(* IEC 61131-3 sources: LabBench/FB, 3 files *)

(* ---- FB_FloatLevelSensorGroup.st ---- *)
(*==============================================================================
    Название:    FB_FloatLevelSensorGroup
    Автор:       Инженер ПЛК
    Дата:        2025-04-26
    Версия:      1.0

    Описание:    Функциональный блок для группы поплавковых датчиков уровня.
                 Группа состоит из трех датчиков, расположенных на различных
                 уровнях в емкости высотой 500 мм:
                 - Нижний: 150 мм
                 - Средний: 250 мм
                 - Верхний: 350 мм

                 Блок обрабатывает сигналы с датчиков, определяет текущий
                 уровень жидкости и проверяет корректность показаний.
==============================================================================*)
FUNCTION_BLOCK FB_FloatLevelSensorGroup
VAR_INPUT
    bLowLevelSensor: BOOL;      (* Сигнал с нижнего датчика (150 мм) *)
    bMidLevelSensor: BOOL;      (* Сигнал со среднего датчика (250 мм) *)
    bHighLevelSensor: BOOL;     (* Сигнал с верхнего датчика (350 мм) *)
    rTankHeightMM: REAL := 500.0; (* Высота емкости, мм *)
    bEnable: BOOL := TRUE;      (* Разрешение работы *)
    bReset: BOOL;               (* Сброс ошибок *)
END_VAR
VAR_OUTPUT
    stData: ST_FloatLevelGroup_Data; (* Структура с результатами *)
END_VAR
VAR
    (* Параметры датчиков *)
    rLowLevelHeightMM: REAL := 150.0;  (* Высота нижнего датчика, мм *)
    rMidLevelHeightMM: REAL := 250.0;  (* Высота среднего датчика, мм *)
    rHighLevelHeightMM: REAL := 350.0; (* Высота верхнего датчика, мм *)

    (* Внутренние переменные *)
    bValid: BOOL;                      (* Флаг валидности данных *)
    bSensorSequenceValid: BOOL;        (* Флаг валидности последовательности *)
END_VAR
VAR CONSTANT
    (* Битовая маска для кодов ошибок *)
    ERR_NONE: WORD := 16#0000;              (* Нет ошибок *)
    ERR_CONFIG: WORD := 16#0001;            (* Ошибка конфигурации *)
    ERR_INVALID_SEQUENCE: WORD := 16#0002;  (* Нарушена последовательность срабатывания *)
    ERR_WIRE_BREAK: WORD := 16#0004;        (* Обрыв линии или неисправность *)
    ERR_SENSOR_FAULT: WORD := 16#0008;      (* Неисправность датчика *)
END_VAR

(* ======================================================================== *)
(* Основная логика функционального блока                                    *)
(* ======================================================================== *)

(* Инициализация *)
stData.bLowLevelActive := FALSE;
stData.bMidLevelActive := FALSE;
stData.bHighLevelActive := FALSE;
stData.wErrorCode := ERR_NONE;
stData.bValid := FALSE;
bValid := FALSE;

(* Проверка конфигурации *)
IF rTankHeightMM <= 0.0 THEN
    (* Некорректно задана высота емкости *)
    stData.eStatus := STATUS_CONFIG_ERROR;
    stData.wErrorCode := stData.wErrorCode OR ERR_CONFIG;

ELSIF rLowLevelHeightMM <= 0.0 OR rMidLevelHeightMM <= 0.0 OR rHighLevelHeightMM <= 0.0 THEN
    (* Некорректно заданы высоты датчиков *)
    stData.eStatus := STATUS_CONFIG_ERROR;
    stData.wErrorCode := stData.wErrorCode OR ERR_CONFIG;

ELSIF rLowLevelHeightMM >= rMidLevelHeightMM OR rMidLevelHeightMM >= rHighLevelHeightMM THEN
    (* Нарушена последовательность высот датчиков *)
    stData.eStatus := STATUS_CONFIG_ERROR;
    stData.wErrorCode := stData.wErrorCode OR ERR_CONFIG;

ELSIF rHighLevelHeightMM >= rTankHeightMM THEN
    (* Верхний датчик выше высоты емкости *)
    stData.eStatus := STATUS_CONFIG_ERROR;
    stData.wErrorCode := stData.wErrorCode OR ERR_CONFIG;

ELSIF NOT bEnable THEN
    (* Блок отключен - возвращаем нулевые значения *)
    stData.eStatus := STATUS_OK;
    stData.rLevelEstimationMM := 0.0;
    stData.rLevelPercent := 0.0;
    stData.wErrorCode := ERR_NONE;
    stData.bValid := FALSE;

ELSE
    (* Нормальная работа - обработка сигналов датчиков *)

    (* Копируем состояния датчиков *)
    stData.bLowLevelActive := bLowLevelSensor;
    stData.bMidLevelActive := bMidLevelSensor;
    stData.bHighLevelActive := bHighLevelSensor;

    (* Проверка последовательности срабатывания датчиков *)
    (* Если верхний датчик активен, средний и нижний тоже должны быть активны *)
    (* Если средний датчик активен, нижний тоже должен быть активен *)
    bSensorSequenceValid := TRUE;

    IF stData.bHighLevelActive AND (NOT stData.bMidLevelActive OR NOT stData.bLowLevelActive) THEN
        (* Верхний датчик активен, но средний или нижний - нет *)
        bSensorSequenceValid := FALSE;
    ELSIF stData.bMidLevelActive AND NOT stData.bLowLevelActive THEN
        (* Средний датчик активен, но нижний - нет *)
        bSensorSequenceValid := FALSE;
    END_IF;

    IF NOT bSensorSequenceValid THEN
        (* Нарушена последовательность срабатывания датчиков *)
        stData.eStatus := STATUS_INVALID_SEQUENCE;
        stData.wErrorCode := stData.wErrorCode OR ERR_INVALID_SEQUENCE;
        bValid := FALSE;
    ELSE
        (* Последовательность корректна - определяем уровень *)
        bValid := TRUE;

        (* Устанавливаем базовый статус *)
        stData.eStatus := STATUS_OK;

        (* Оценка уровня на основе активных датчиков *)
        IF stData.bHighLevelActive THEN
            (* Все три датчика активны - высокий уровень *)
            stData.rLevelEstimationMM := rHighLevelHeightMM;
        ELSIF stData.bMidLevelActive THEN
            (* Активны нижний и средний датчики - средний уровень *)
            stData.rLevelEstimationMM := rMidLevelHeightMM;
        ELSIF stData.bLowLevelActive THEN
            (* Активен только нижний датчик - низкий уровень *)
            stData.rLevelEstimationMM := rLowLevelHeightMM;
        ELSE
            (* Ни один датчик не активен - уровень ниже нижнего датчика *)
            stData.rLevelEstimationMM := rLowLevelHeightMM / 2.0; (* Примерная оценка - половина высоты нижнего датчика *)
        END_IF;

        (* Расчет процентного значения от максимальной высоты *)
        IF rTankHeightMM > 0.0 THEN
            stData.rLevelPercent := (stData.rLevelEstimationMM / rTankHeightMM) * 100.0;
        ELSE
            stData.rLevelPercent := 0.0;
        END_IF;
    END_IF;

    (* Установка флага валидности *)
    stData.bValid := bValid;
END_IF;

(* Сброс ошибок по внешнему сигналу *)
IF bReset THEN
    stData.eStatus := STATUS_OK;
    stData.wErrorCode := ERR_NONE;
    stData.bValid := TRUE;
END_IF;

(* ---- FB_FlowSensor.st ---- *)
(*==============================================================================
    Название:    FB_FlowSensor
    Автор:       Редько А.
    Дата:        2025-04-27
    Версия:      1.0

    Описание:    Универсальный функциональный блок для расходомеров
                 с частотным/импульсным выходом.
==============================================================================*)
FUNCTION_BLOCK FB_FlowSensor
VAR_INPUT
    wPulseCounter: WORD;          (* Значение счетчика импульсов *)
    rPulsePerLiter: REAL;         (* Количество импульсов на литр *)
    tSampleTime: TIME := T#500MS; (* Время выборки для расчета расхода *)
    bEnable: BOOL := TRUE;        (* Разрешение работы *)
    bReset: BOOL;                 (* Сброс счетчиков и ошибок *)
END_VAR
VAR_OUTPUT
    stData: ST_FlowSensor_Data;   (* Структура с результатами *)
END_VAR
VAR
    (* Переменные для обработки импульсов *)
    dwPrevPulseCount: DWORD;      (* Предыдущее значение счетчика импульсов *)
    dwCurrentPulseCount: DWORD;   (* Текущее значение счетчика импульсов *)
    dwTotalPulseCount: DWORD;     (* Общее количество импульсов с учетом переполнений *)
    dwOverflowCounter: DWORD;     (* Счетчик переполнений WORD *)

    bFirstCycle: BOOL := TRUE;    (* Флаг первого цикла *)
    bValid: BOOL;                 (* Флаг валидности данных *)

    tTimer: TON;                  (* Таймер для расчета расхода *)
    rSampleTimeInSec: REAL;       (* Время выборки в секундах *)
END_VAR
VAR CONSTANT
    (* Битовая маска для кодов ошибок *)
    ERR_NONE: WORD := 16#0000;            (* Нет ошибок *)
    ERR_CONFIG: WORD := 16#0001;          (* Ошибка конфигурации *)
END_VAR

(* ======================================================================== *)
(* Основная логика функционального блока                                    *)
(* ======================================================================== *)

(* Инициализация *)

stData.wErrorCode := ERR_NONE;
stData.bValid := FALSE;
bValid := FALSE;

(* Проверка конфигурации *)
IF rPulsePerLiter <= 0.0 THEN
    (* Некорректно задан коэффициент пересчета *)
    stData.eStatus := STATUS_CONFIG_ERROR;
    stData.wErrorCode := stData.wErrorCode OR ERR_CONFIG;

ELSIF NOT bEnable THEN
    (* Блок отключен - нулевые значения *)
    stData.eStatus := STATUS_OK;
    stData.rFlowLPM := 0.0;
    stData.rFlowM3H := 0.0;
    stData.rFrequencyHz := 0.0;
    stData.wErrorCode := ERR_NONE;
    stData.bValid := FALSE;

ELSE
    (* Нормальная работа - обработка данных *)

    (* Преобразование WORD в DWORD *)
    dwCurrentPulseCount := WORD_TO_DWORD(wPulseCounter); (*  *)

    (* Обработка первого вызова *)
    IF bFirstCycle THEN
        dwPrevPulseCount := dwCurrentPulseCount;
        dwTotalPulseCount := dwCurrentPulseCount;
        bFirstCycle := FALSE; (*  *)
    END_IF;

    (* Обработка переполнения счетчика *)
    IF dwCurrentPulseCount < dwPrevPulseCount THEN
        (* Счетчик переполнился - добавляем 65536 (2^16) *)
        dwOverflowCounter := dwOverflowCounter + 65536;
    END_IF;

    (* Расчет общего количества импульсов *)
    dwTotalPulseCount := dwCurrentPulseCount + dwOverflowCounter;
    stData.dwPulseCount := dwTotalPulseCount;

    (* Запуск таймера для расчета расхода *)
    tTimer(IN := TRUE, PT := tSampleTime);

    (* Расчет расхода по частоте импульсов *)
    IF tTimer.Q THEN
        (* Вычисление количества импульсов за период *)
        stData.dwPulseDelta := dwTotalPulseCount - dwPrevPulseCount;
        dwPrevPulseCount := dwTotalPulseCount;

        (* Преобразование времени выборки в секунды *)
        rSampleTimeInSec := TIME_TO_REAL(tSampleTime) / 1000.0;

        (* Расчет частоты импульсов (Гц) *)
        stData.rFrequencyHz := DWORD_TO_REAL(stData.dwPulseDelta) / rSampleTimeInSec;

        (* Расчет расхода в л/мин - универсальная формула для любого расходомера *)
        stData.rFlowLPM := (stData.rFrequencyHz * 60.0) / rPulsePerLiter;

        (* Расчет расхода в м?/ч *)
        stData.rFlowM3H := stData.rFlowLPM * 0.06; (* 1 л/мин = 0.06 м?/ч *)

        (* Расчет общего объема в литрах (полезно для учебных целей) *)
        stData.rTotalLiters := DWORD_TO_REAL(stData.dwPulseCount) / rPulsePerLiter;

        ⁡⁢⁣⁣(* Данные валидны *)⁡
        bValid := TRUE;
        stData.eStatus := STATUS_OK;

        (* Сброс таймера для следующего периода *)
        tTimer(IN := FALSE);
    END_IF;

    (* Установка флага валидности *)
    stData.bValid := bValid;
END_IF;

(* Сброс по внешнему сигналу *)
IF bReset THEN
    dwPrevPulseCount := dwCurrentPulseCount;
    dwOverflowCounter := 0;
    stData.rTotalLiters := 0.0;
    stData.eStatus := STATUS_OK;
    stData.wErrorCode := ERR_NONE;
    stData.bValid := TRUE;
END_IF;

(* ---- FB_PressureSensor.st ---- *)
(*==============================================================================
    Название:    FB_PressureSensor
    Автор:       Редько А.
    Дата:        2025-04-25
    Версия:      1.1

    Описание:    Функциональный блок для датчиков давления.

                 Данные получаются после масштабирования в конфигурации ПЛК.
                 Блок проверяет статус измерения, выполняет проверку на
                 превышение предельного значения и формирует структуру данных
                 с результатами.

    Примечание:  Фильтрация и обработка статусов выполняется в конфигурации ПЛК
==============================================================================*)
FUNCTION_BLOCK FB_PressureSensor
VAR_INPUT
    rPressureKPa: REAL;         (* Давление в кПа (с аналогового входа после масштабирования) *)
    rMaxPressureKPa: REAL;      (* Максимально допустимое давление, кПа *)
    bEnable: BOOL := TRUE;      (* Разрешение работы *)
    bReset: BOOL;               (* Сброс ошибок *)
END_VAR

VAR_OUTPUT
    stData: ST_PressureSensor_Data;  (* Структура с результатами *)
END_VAR

VAR
    (* Системные переменные *)
    byStatus: BYTE;              (* Старший байт из переменной для анализа статуса *)
    bValid: BOOL;                 (* Флаг валидности данных *)
END_VAR

VAR CONSTANT
    (* Константы для статусов аналогового входа (старший байт) *)
    ERR_NONE: BYTE := 16#00;           (* Ошибок нет *)
    ERR_INVALID: BYTE := 16#F1;        (* Результаты измерения заведомо неверны *)
    ERR_NOT_READY: BYTE := 16#F6;      (* Результаты измерения не готовы *)
    ERR_ABOVE_RANGE: BYTE := 16#FA;    (* Сигнал на входе больше возможного *)
    ERR_BELOW_RANGE: BYTE := 16#FB;    (* Сигнал на входе меньше возможного *)
    ERR_CURRENT_OVERLOAD: BYTE := 16#FC;(* Перегрузка в канале измерения тока *)
    ERR_VOLTAGE_BREAK: BYTE := 16#FD;  (* Обрыв датчика в канале измерения напряжения *)

    (* Битовые маски для кодов ошибок *)
    ERROR_NONE: WORD := 16#0000;           (* Нет ошибок *)
    ERROR_CONFIG: WORD := 16#0001;         (* Ошибка конфигурации *)
    ERROR_VALUE_ABOVE_MAX: WORD := 16#0002;    (* Превышение максимального давления *)
    ERROR_AI_ABOVE_RANGE: WORD := 16#0004; (* Превышение диапазона аналогового входа *)
    ERROR_AI_BELOW_RANGE: WORD := 16#0008; (* Значение ниже диапазона аналогового входа *)
    ERROR_WIRE_BREAK: WORD := 16#0010;     (* Обрыв линии датчика *)
    ERROR_CURRENT_OVERLOAD: WORD := 16#0020; (* Перегрузка в канале измерения тока *)
    ERROR_NOT_READY: WORD := 16#0040;      (* Измерение не готово *)
    ERROR_UNKNOWN: WORD := 16#8000;        (* Неизвестная ошибка *)
END_VAR

(* ======================================================================== *)
(* Основная логика функционального блока                                    *)
(* ======================================================================== *)

(* Инициализация *)
stData.rPressureKPa := rPressureKPa;  (* Сохраняем исходное значение *)
stData.wErrorCode := ERROR_NONE;
stData.bValid := FALSE;
bValid := FALSE;

(* Проверка конфигурации *)
IF rMaxPressureKPa <= 0.0 THEN
    (* Некорректно задано максимальное давление *)
    stData.eStatus := STATUS_CONFIG_ERROR;
    stData.wErrorCode := stData.wErrorCode OR ERROR_CONFIG;

ELSIF NOT bEnable THEN
    (* Блок отключен - возвращаем нулевые значения *)
    stData.eStatus := STATUS_OK;
    stData.rPressureKPa := 0.0;
    stData.wErrorCode := ERROR_NONE;
    stData.bValid := FALSE;

ELSE
    (* Нормальная работа - обработка данных и проверка ошибок *)

    (* Получение старшего байта для анализа статуса *)
    byStatus := DWORD_TO_BYTE(SHR(REAL_TO_DWORD(rPressureKPa) AND 16#FF000000, 24));

    (* Проверка статуса аналогового входа *)
    CASE byStatus OF
        ERR_NONE:
            (* Нормальные данные - статус OK *)
            stData.eStatus := STATUS_OK;
            bValid := TRUE;

        ERR_ABOVE_RANGE:
            (* Превышение диапазона аналогового входа *)
            stData.eStatus := STATUS_AI_ABOVE_RANGE;
            stData.wErrorCode := stData.wErrorCode OR ERROR_AI_ABOVE_RANGE;
            bValid := FALSE;

        ERR_BELOW_RANGE:
            (* Значение ниже диапазона аналогового входа *)
            stData.eStatus := STATUS_AI_BELOW_RANGE;
            stData.wErrorCode := stData.wErrorCode OR ERROR_AI_BELOW_RANGE;
            bValid := FALSE;

        ERR_VOLTAGE_BREAK:
            (* Обрыв линии датчика *)
            stData.eStatus := STATUS_WIRE_BREAK;
            stData.wErrorCode := stData.wErrorCode OR ERROR_WIRE_BREAK;
            bValid := FALSE;

        ERR_CURRENT_OVERLOAD:
            (* Перегрузка в канале измерения тока *)
            stData.eStatus := STATUS_CURRENT_OVERLOAD;
            stData.wErrorCode := stData.wErrorCode OR ERROR_CURRENT_OVERLOAD;
            bValid := FALSE;

        ERR_NOT_READY:
            (* Измерение не готово *)
            stData.eStatus := STATUS_NOT_READY;
            stData.wErrorCode := stData.wErrorCode OR ERROR_NOT_READY;
            bValid := FALSE;

        ELSE
            (* Прочие неизвестные ошибки *)
            stData.eStatus := STATUS_UNKNOWN;
            stData.wErrorCode := stData.wErrorCode OR ERROR_UNKNOWN;
            bValid := FALSE;
    END_CASE;

    (* Проверка на превышение максимально допустимого давления *)
    IF rPressureKPa > rMaxPressureKPa AND rMaxPressureKPa > 0.0 AND bValid THEN
        (* Выставляем ошибку превышения давления *)
        stData.eStatus := STATUS_VALUE_ABOVE_MAX;
        stData.wErrorCode := stData.wErrorCode OR ERROR_VALUE_ABOVE_MAX;
        bValid := FALSE;
    END_IF;

    (* Установка флага валидности *)
    stData.bValid := bValid;
END_IF;

(* Сброс ошибок по внешнему сигналу *)
IF bReset THEN
    stData.eStatus := STATUS_OK;
    stData.wErrorCode := ERROR_NONE;
    stData.bValid := TRUE;
END_IF;
